Fanuc KAREL source: kt00564.KL

-- PROVISIONAL review KL for V770-1; original PC SHA256 fcada62e8f90855dd94d6f92e0e13f993f65c3db1d3f44b6e9a747205b64f5b0
-- Incomplete behavior may be omitted. Consult companion uncertainty JSON. Do not deploy.
PROGRAM KT00564
%NOLOCKGROUP
VAR
  OUT : REAL
-- UNRESOLVED_DECL V1 type=000013
-- UNRESOLVED_DECL V2 type=000013
BEGIN
  -- UNRESOLVED_PC offsets 5-20; opcodes 2E,22,32,35
  -- UNRESOLVED_PC offsets 25-40; opcodes 2E,22,32,35
  -- UNRESOLVED_PC offsets 45-60; opcodes 2E,22,32,35
  -- UNRESOLVED_PC offsets 65-80; opcodes 2E,22,32,35
  -- UNRESOLVED_PC offsets 85-108; opcodes 49,49,94,23
  -- UNRESOLVED_PC offsets 113-117; opcodes 7F
END KT00564
